TYPE ST_ProductionData_HMI :
    STRUCT
        bHMIControlAvailable    : BOOL; //Set TRUE *FROM PLC* when HMI requests can be processed
        bIncomingHMIRequest     : BOOL; //Pulses TRUE when an HMI request is issued
        bHMICommandConfirmation : BOOL; //Confirms receipt and subsequent processing of the command sent by the HMI

        bShiftLengthHMISetRequest : BOOL;
        tShiftLengthHMISetValue   : TIME;

        bShiftProductionTargetHMISetRequest : BOOL;
        nShiftProductionTargetHMISetValue   : DINT;

        bWarningMarginHMISetRequest : BOOL;
        fWarningMarginHMISetValue   : LREAL;

        bProductionRateHMISetRequest : BOOL;
        fProductionRateHMISetValue   : LREAL;

        tShiftLength           : TIME; //Specify the time duration of a shift
        nShiftProductionTarget : DINT; //Specify the desired production count by end of shift

        nCurrentAcceptableProductionCount : DINT;
        nCurrentWarningProductionCount    : DINT;
        nCurrentShiftProductionCount      : DINT; //Number of products completed so far on the current shift
        nCurrentShiftTarget               : DINT; //Expected number of completed products at the current time in the shift
        tCurrentShiftTime                 : TIME; //Time elapsed since the start of the shift
        tRemainingShiftTime               : TIME; //Time remaining in the current shift
        tShiftStartTimeStamp              : TIMESTRUCT;
        tShiftStartTimeStamp_UTC          : STRING;
        fProductionRate_Setpoint          : LREAL;
        fProductionRate_Actual            : LREAL;
        fProductionRate_Required          : LREAL;

    END_STRUCT
END_TYPE

(* stored: Version 1.1.0.1, ProductVersion 3.1.4024.11
   DUT ST_ProductionData_HMI: Id {bc82133b-7334-4077-94d6-923513c1c9b1} *)
